TYPE T_PAYLOAD :
STRUCT
	data1 : LREAL := 1.51; 
	data2 : LREAL := 12345.122; 
END_STRUCT
END_TYPE

(* stored: Version 1.1.0.1, ProductVersion 3.1.4024.9
   DUT T_PAYLOAD: Id {ba34a113-6e0b-4b76-9937-93a1c84b842b} *)
